PROGRAM MAIN
VAR
	bStart : BOOL;
	bRunning : BOOL;
END_VAR

IF bStart THEN
	bRunning := TRUE;
ELSE
	bRunning := FALSE;
END_IF

END_PROGRAM

(* stored: Version 1.1.0.1, ProductVersion 3.1.4024.16
   POU MAIN: Id {fbcf839e-58f6-4279-ae35-e59b3861a9d2}, SpecialFunc None *)
